PROGRAM main
  VAR_EXTERNAL
    TEMP_ALARM : BOOL;
  END_VAR
  VAR
    START_PB : BOOL;
    MOTOR_RUN : BOOL;
    STOP_PB : BOOL;
    MOTOR_VOLTAGE : INT := 380; (* MOTOR VOLTAGE [V] *)
    MOTOR_CURRENT : REAL := 12.5; (* MOTOR CURRENT [A] *)
  END_VAR

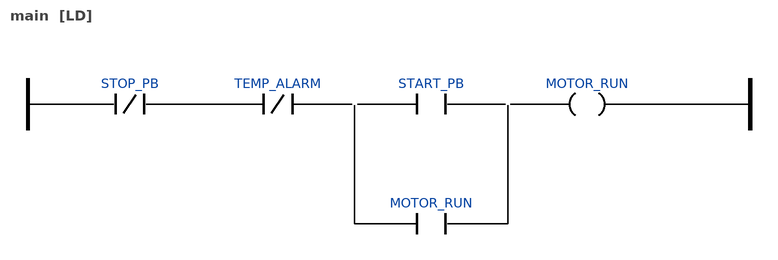
(* LD diagram, written out as Structured Text *)
MOTOR_RUN := NOT STOP_PB AND NOT TEMP_ALARM AND (START_PB OR MOTOR_RUN);
END_PROGRAM
